INTERFACE I_ActuatorBase EXTENDS __System.IQueryInterface

{attribute 'monitoring' := 'call'}
PROPERTY public inError : bool
GET
END_GET
END_PROPERTY

{attribute 'monitoring' := 'call'}
PROPERTY public isBusy : bool
GET
END_GET
END_PROPERTY

{attribute 'monitoring' := 'call'}
PROPERTY public isOff : BOOL
GET
END_GET
END_PROPERTY

{attribute 'monitoring' := 'call'}
PROPERTY public noFeed : BOOL
GET
END_GET
END_PROPERTY

{attribute 'monitoring' := 'call'}
PROPERTY public ok : bool
GET
END_GET
END_PROPERTY

METHOD PUBLIC reset : BOOL
VAR_INPUT
END_VAR
END_METHOD

METHOD public switchOff : BOOL
VAR_INPUT
END_VAR
END_METHOD

END_INTERFACE

(* stored: Version 1.1.0.1, ProductVersion 3.1.4024.3
   Itf I_ActuatorBase: Id {46dad2fc-156d-45ec-93cd-344afa0e6051}
   Property inError: Id {d2f5904c-cc87-4105-a9ee-d5febb327cf7}
   Get Get: Id {f7ebf349-22c4-4344-9d9f-bbc02e053d44}
   Property isBusy: Id {b869e0fc-662e-4f15-91cc-14948c70232d}
   Get Get: Id {14abb90e-d9ee-4282-9ae1-3b596128d2c7}
   Property isOff: Id {31bd977b-7f66-404d-a919-f85ff3bd7c66}
   Get Get: Id {56c493d5-9a94-40a7-9b0c-b47bb6e395df}
   Property noFeed: Id {042ef271-dd59-4c9f-bf93-8dcb09222e48}
   Get Get: Id {0e95e137-8fcb-41b8-8897-ab3694c157a4}
   Property ok: Id {831fa375-e8a7-4c6b-affd-d8044e891d10}
   Get Get: Id {1a37b8a3-e8e4-49bc-8b96-6f5f7181c205}
   Method reset: Id {b89a9eb2-a357-408f-8267-532cdc90d8e2}
   Method switchOff: Id {de37676c-e8e3-41b4-b62d-9df26640547f} *)
